SYSTEM TEST_SELA (* Test FB_SEL_ARRAY *)
  (* Standard: 61499-1 *)
  (* Version 0.0, 2006-09-13, JHC, Holobloc Inc *)
  DEVICE DEV1 : FRAME_DEVICE(BOUNDS := [100,100,100,150], GRID := [1,1])
    RESOURCE RES1 : PANEL_RESOURCE(ROWS := 4, COLS := 1)
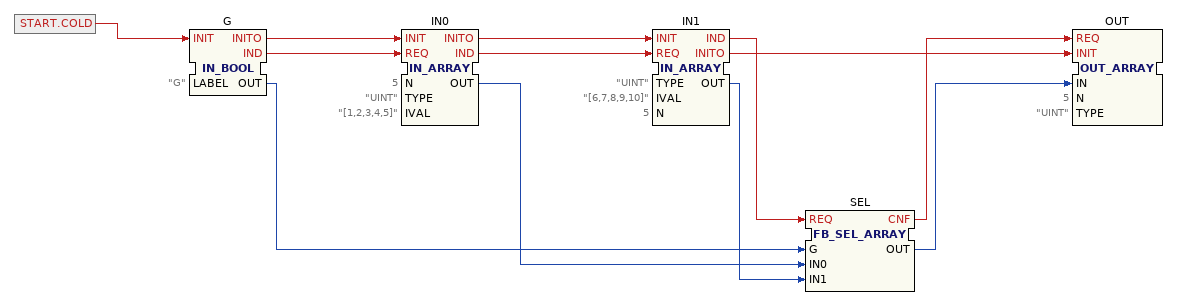
      FBS
        G : IN_BOOL(LABEL := "G");
        IN0 : IN_ARRAY(N := 5, TYPE := "UINT", IVAL := "[1,2,3,4,5]");
        IN1 : IN_ARRAY(TYPE := "UINT", IVAL := "[6,7,8,9,10]", N := 5);
        SEL : FB_SEL_ARRAY;
        OUT : OUT_ARRAY(N := 5, TYPE := "UINT");
      END_FBS
      EVENT_CONNECTIONS
        G.INITO TO IN0.INIT;
        START.COLD TO G.INIT;
        G.IND TO IN0.REQ;
        IN0.INITO TO IN1.INIT;
        IN0.IND TO IN1.REQ;
        IN1.IND TO SEL.REQ;
        SEL.CNF TO OUT.REQ;
        IN1.INITO TO OUT.INIT;
      END_CONNECTIONS
      DATA_CONNECTIONS
        G.OUT TO SEL.G;
        IN0.OUT TO SEL.IN0;
        IN1.OUT TO SEL.IN1;
        SEL.OUT TO OUT.IN;
      END_CONNECTIONS
    END_RESOURCE
  END_DEVICE
END_SYSTEM
